// TwinCAT 3 PLC project GenevaTest
// ProgramVersion: 3.1.4020.4
// libraries:
//   Tc2_MC2, * (Beckhoff Automation GmbH)
//   Tc2_Standard, * (Beckhoff Automation GmbH)
//   Tc2_System, * (Beckhoff Automation GmbH)
//   Tc3_Module, * (Beckhoff Automation GmbH)
// project tree:
//   / PlcTask.TcTTO
//   POUs/ MAIN.TcPOU
// real-time tasks:
//   TASK PlcTask: cycle T#10ms, priority 20, ADS port 350
// motion (NC):
// I/O:
//   DEVICE Device 1 (EtherCAT), AmsNetId 5.45.6.154.2.1
//     Term 1 (EK1200) [EK1200-5000 EtherCAT Power supply (2A E-Bus)]
//       Term 2 (EL7031)
//       Term 3 (EL7041)
//       Term 4 (EL5042)
//       Term 5 (EL1004) [EL1004 4Ch. Dig. Input 24V, 3ms]
//       Term 6 (EL2008) [EL2008 8Ch. Dig. Output 24V, 0.5A]
//       Term 7 (EL9011) [EL9011 End Terminal]
// variable links:
//   GenevaTest Instance <-> Device 1 (EtherCAT)/Term 1 (EK1200)/Term 2 (EL7031)
//     PlcTask Inputs/MAIN.bLimBwd2 <-> STM Status/Status/Digital input 2
//     PlcTask Inputs/MAIN.bLimFwd2 <-> STM Status/Status/Digital input 1
//   GenevaTest Instance <-> Device 1 (EtherCAT)/Term 1 (EK1200)/Term 6 (EL2008)
//     PlcTask Outputs/MAIN.bBrake2 <-> Channel 1/Output
//   GenevaTest Instance <-> NC-Task 1 SAF/Axes/Axis 1
//     PlcTask Inputs/MAIN.axis1.NcToPlc <-> Outputs/ToPlc
//     PlcTask Outputs/MAIN.axis1.PlcToNc <-> Inputs/FromPlc
//   GenevaTest Instance <-> NC-Task 1 SAF/Axes/Axis 2
//     PlcTask Inputs/MAIN.axis2.NcToPlc <-> Outputs/ToPlc
//     PlcTask Outputs/MAIN.axis2.PlcToNc <-> Inputs/FromPlc

CONFIGURATION GenevaTest
    RESOURCE PLC ON TwinCAT3
        TASK PlcTask(INTERVAL := T#10ms, PRIORITY := 20);
        PROGRAM MAIN WITH PlcTask : MAIN;
    END_RESOURCE
END_CONFIGURATION

// ---- POUs/MAIN.TcPOU
PROGRAM MAIN
VAR
	fbPower1: MC_POWER;
	axis1: AXIS_REF;
	fbPower2: MC_POWER;
	axis2: AXIS_REF;
	bLimFwd2 AT %I*: BOOL;
	bLimBwd2 AT %I*: BOOL;
	bBrake2 AT %Q*: BOOL;
END_VAR

axis1.ReadStatus();
fbPower1(Axis:=axis1,
	Enable:=TRUE,
	Enable_Positive:=TRUE,
	Enable_Negative:=TRUE);
axis2.ReadStatus();
fbPower2(Axis:=axis2,
	Enable:=TRUE,
	Enable_Positive:=bLimFwd2,
	Enable_Negative:=bLimBwd2);
bBrake2 := axis2.Status.ControlLoopClosed;

END_PROGRAM
